TEXTLIST KPickMode
  0 = 'Suction'
  1 = 'Position'
  2 = 'Position+Torque'
   = ''
END_TEXTLIST

(* stored: Version 1.1.0.1, ProductVersion 3.1.4024.11
   TextList KPickMode: Id {a5eb016b-dcc9-4eb9-ad72-0fccee03c9b4} *)
